# EPICS substitutions: db/ecmcEL9410.substitutions
file ecmcEcSlave.template
{
    pattern {}
            {}
}

file ecmcEL9410.template
{
	pattern {}
		    {}
}
